# EPICS substitutions: PIP-II/RFPI2/rfpi-fdr-sw-mgmt-ioc-main/ina-managementApp/Db/fan.substitutions
file fan.template {
pattern{ acc, sys, group, num, fan_idx }
{ PIP2IT, pHB650, RFPI, ina, 1 }
{ PIP2IT, pHB650, RFPI, ina, 2 }
{ PIP2IT, pHB650, RFPI, ina, 3 }
}
